PROGRAM MAIN
VAR
	nCounter 				: INT;
	fbTestSimpleDynBuffer 	: FB_TestSimpleDynBuffer;
	fbTestVarByteBuffer		: FB_TestVarStringBuffer;
END_VAR

nCounter := nCounter + 1;

TcUnit.RUN();

END_PROGRAM

(* stored: Version 1.1.0.1
   POU MAIN: Id {7ced7848-7e71-4263-9269-881b93844670}, SpecialFunc None *)
